TYPE InputBase_8311D824 :
STRUCT
END_STRUCT
END_TYPE

(* stored: Version 1.2.0.0, ProductVersion 3.1.4024.9
   DUT InputBase_8311D824: Id {c4a56999-ad48-4395-b06f-46c701784849} *)
